FUNCTION F_StrategyFunction : I_FillingStrategy
VAR_INPUT
	stBottle : REFERENCE TO ST_Bottle;
END_VAR

VAR
	fbHoneyFill : FB_HoneyFill;
END_VAR

CASE stBottle.eLiquidType OF
	E_LiquidType.HONEY:
	F_StrategyFunction := fbHoneyFill;
	
	E_LiquidType.SODA:
	F_StrategyFunction := GVL_References.g_fbSodaFill;
	
	E_LiquidType.WATER:
	F_StrategyFunction := GVL_References.g_fbWaterFill;
END_CASE

END_FUNCTION

(* stored: Version 1.1.0.1, ProductVersion 3.1.4024.16
   POU F_StrategyFunction: Id {2efe749e-a201-4d1b-96b2-96e98e0e450f}, SpecialFunc None *)
